// TIA Portal V17 export
// export: Created 2022-06-27T13:57:44.2303168Z, ExportSetting WithDefaults, DisplayName Totally Integrated Automation Portal, DisplayVersion V17 Update 3, DisplayName TIA Portal Openness, DisplayVersion V17 Update 3, DisplayName TIA Portal Version Control Interface, DisplayVersion V17, DisplayName SINAMICS Startdrive Advanced, DisplayVersion V17 Update1, DisplayName SINAMICS Startdrive G110M, G120, G120C, G120D, G120P, G115D, DisplayVersion V17 Update1, DisplayName SINAMICS Startdrive G130, G150, S120, S150, SINAMICS MV, S210, DisplayVersion V17 Update1, DisplayName STEP 7 Professional, DisplayVersion V17 Update 3, DisplayName STEP 7 Safety, DisplayVersion V17, DisplayName WinCC UA Professional, DisplayVersion V17 Update 3
FUNCTION_BLOCK "S041_DIRECT_START_MOTOR"   // FB41, LAD
{ S7_Optimized_Access := 'TRUE' }
VERSION : 0.1
// Info:
// -Motors that are named "Uxx-xx" instead of "Mxx-xx" use soft-starters
// stored: AutoNumber false, IsIECCheckEnabled false, IsRetainMemResEnabled false, MemoryReserve 100, SetENOAutomatically false, UDAEnableTagReadback false
   VAR
      ls_aDirect_Start_Motors : Bool;
      ls_aDriver_Motors : Bool;
      FB_INTERLOCKS_U33_2D { S7_SetPoint := 'True'} : "FB_INTERLOCKS";
      FB_MOTOR_DIRECT_START_U33_2D { S7_SetPoint := 'True'} : "FB_MOTOR_DIRECT_START";
      FB_INTERLOCKS_M33_4F { S7_SetPoint := 'True'} : "FB_INTERLOCKS";
      FB_MOTOR_DIRECT_START_M33_4F { S7_SetPoint := 'True'} : "FB_MOTOR_DIRECT_START";
      FB_INTERLOCKS_M33_6F { S7_SetPoint := 'True'} : "FB_INTERLOCKS";
      FB_MOTOR_DIRECT_START_M33_6F { S7_SetPoint := 'True'} : "FB_MOTOR_DIRECT_START";
      FB_INTERLOCKS_M35_2D { S7_SetPoint := 'True'} : "FB_INTERLOCKS";
      FB_MOTOR_DIRECT_START_M35_2D { S7_SetPoint := 'True'} : "FB_MOTOR_DIRECT_START";
      FB_MOTOR_DIRECT_START_U35_4D { S7_SetPoint := 'True'} : "FB_MOTOR_DIRECT_START";
      FB_INTERLOCKS_M36_5F { S7_SetPoint := 'True'} : "FB_INTERLOCKS";
      FB_MOTOR_DIRECT_START_M36_5F { S7_SetPoint := 'True'} : "FB_MOTOR_DIRECT_START";
      FB_INTERLOCKS_M36_7F { S7_SetPoint := 'True'} : "FB_INTERLOCKS";
      FB_MOTOR_DIRECT_START_M36_7F { S7_SetPoint := 'True'} : "FB_MOTOR_DIRECT_START";
      FB_INTERLOCKS_M36_9F { S7_SetPoint := 'True'} : "FB_INTERLOCKS";
      FB_MOTOR_DIRECT_START_M36_9F { S7_SetPoint := 'True'} : "FB_MOTOR_DIRECT_START";
      FB_INTERLOCKS_U37_2D { S7_SetPoint := 'True'} : "FB_INTERLOCKS";
      FB_MOTOR_DIRECT_START_U37_2D { S7_SetPoint := 'True'} : "FB_MOTOR_DIRECT_START";
      FB_INTERLOCKS_U37_3D { S7_SetPoint := 'True'} : "FB_INTERLOCKS";
      FB_MOTOR_DIRECT_START_U37_3D { S7_SetPoint := 'True'} : "FB_MOTOR_DIRECT_START";
      FB_INTERLOCKS_M37_5F { S7_SetPoint := 'True'} : "FB_INTERLOCKS";
      FB_MOTOR_DIRECT_START_M37_5F { S7_SetPoint := 'True'} : "FB_MOTOR_DIRECT_START";
      FB_INTERLOCKS_M37_7F { S7_SetPoint := 'True'} : "FB_INTERLOCKS";
      FB_MOTOR_DIRECT_START_M37_7F { S7_SetPoint := 'True'} : "FB_MOTOR_DIRECT_START";
      FB_INTERLOCKS_M37_9F { S7_SetPoint := 'True'} : "FB_INTERLOCKS";
      FB_MOTOR_DIRECT_START_M37_9F { S7_SetPoint := 'True'} : "FB_MOTOR_DIRECT_START";
      FB_INTERLOCKS_U35_4D { S7_SetPoint := 'True'} : "FB_INTERLOCKS";
   END_VAR
BEGIN

REGION Network 1: U33-2D - Burner Fan - Automatic on and off
END_REGION

REGION Network 2: U33-2D - Burner Fan - Interlocks
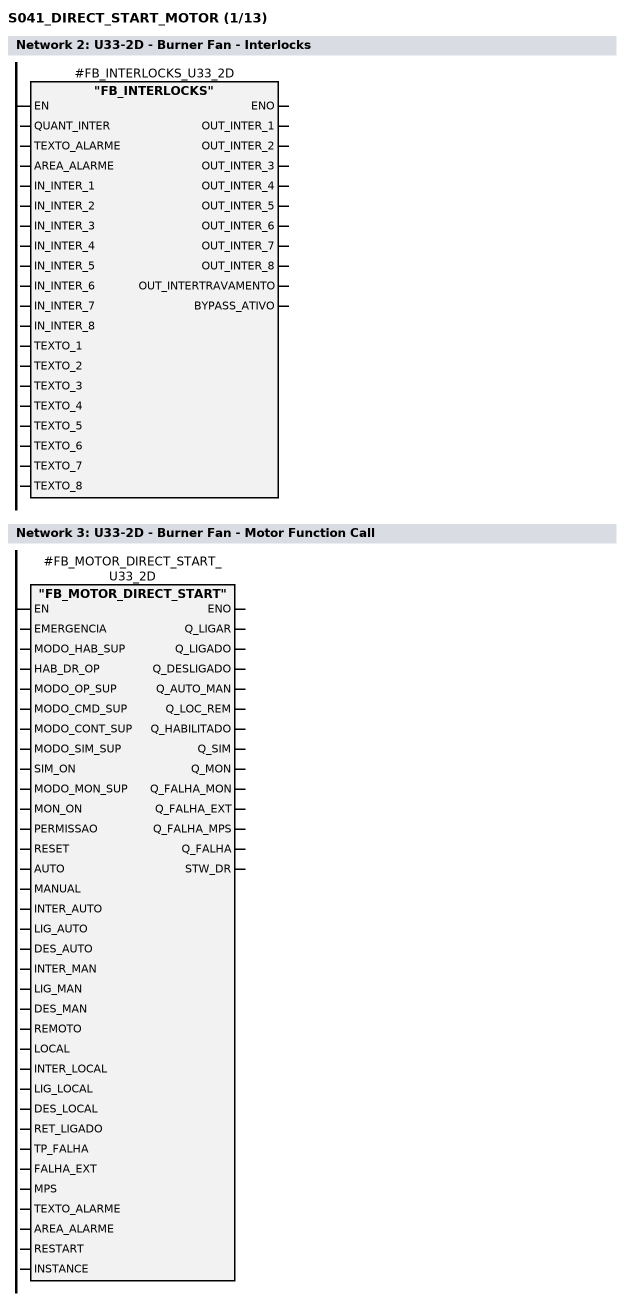
   RUNG wire#powerrail
      #FB_INTERLOCKS_U33_2D(QUANT_INTER :=, TEXTO_ALARME :=, AREA_ALARME :=, IN_INTER_1 :=, IN_INTER_2 :=, IN_INTER_3 :=, IN_INTER_4 :=, IN_INTER_5 :=, IN_INTER_6 :=, IN_INTER_7 :=, IN_INTER_8 :=, TEXTO_1 :=, TEXTO_2 :=, TEXTO_3 :=, TEXTO_4 :=, TEXTO_5 :=, TEXTO_6 :=, TEXTO_7 :=, TEXTO_8 :=, OUT_INTER_1 =>, OUT_INTER_2 =>, OUT_INTER_3 =>, OUT_INTER_4 =>, OUT_INTER_5 =>, OUT_INTER_6 =>, OUT_INTER_7 =>, OUT_INTER_8 =>, OUT_INTERTRAVAMENTO =>, BYPASS_ATIVO =>)
   END_RUNG
   // the same network as SCL:
   #FB_INTERLOCKS_U33_2D();   // "FB_INTERLOCKS"
END_REGION

REGION Network 3: U33-2D - Burner Fan - Motor Function Call
   RUNG wire#powerrail
      #FB_MOTOR_DIRECT_START_U33_2D(EMERGENCIA :=, MODO_HAB_SUP :=, HAB_DR_OP :=, MODO_OP_SUP :=, MODO_CMD_SUP :=, MODO_CONT_SUP :=, MODO_SIM_SUP :=, SIM_ON :=, MODO_MON_SUP :=, MON_ON :=, PERMISSAO :=, RESET :=, AUTO :=, MANUAL :=, INTER_AUTO :=, LIG_AUTO :=, DES_AUTO :=, INTER_MAN :=, LIG_MAN :=, DES_MAN :=, REMOTO :=, LOCAL :=, INTER_LOCAL :=, LIG_LOCAL :=, DES_LOCAL :=, RET_LIGADO :=, TP_FALHA :=, FALHA_EXT :=, MPS :=, TEXTO_ALARME :=, AREA_ALARME :=, RESTART :=, INSTANCE :=, Q_LIGAR =>, Q_LIGADO =>, Q_DESLIGADO =>, Q_AUTO_MAN =>, Q_LOC_REM =>, Q_HABILITADO =>, Q_SIM =>, Q_MON =>, Q_FALHA_MON =>, Q_FALHA_EXT =>, Q_FALHA_MPS =>, Q_FALHA =>, STW_DR =>)
   END_RUNG
   // the same network as SCL:
   #FB_MOTOR_DIRECT_START_U33_2D();   // "FB_MOTOR_DIRECT_START"
END_REGION

REGION Network 4: U33-2D - Burner Fan - Circuit Breaker
END_REGION

REGION Network 6: M33-4F - Rotary Valve Roaster Cyclone - Automatic on and off
END_REGION

REGION Network 7: M33-4F - Rotary Valve Roaster Cyclone - Interlocks
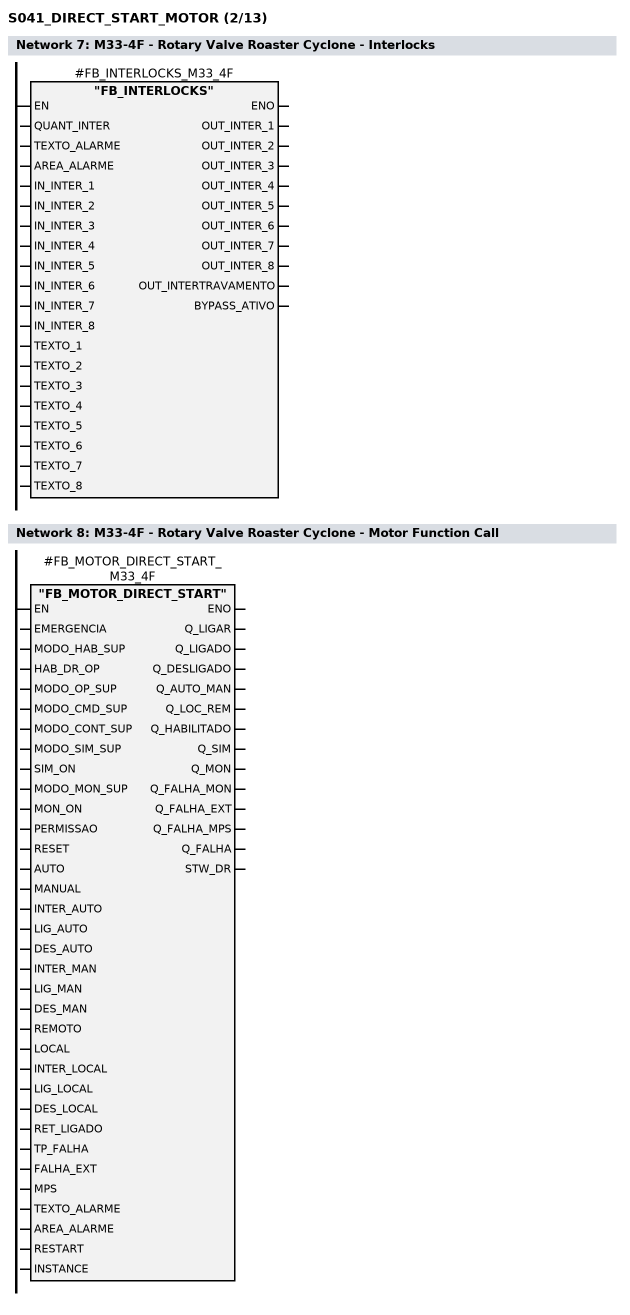
   RUNG wire#powerrail
      #FB_INTERLOCKS_M33_4F(QUANT_INTER :=, TEXTO_ALARME :=, AREA_ALARME :=, IN_INTER_1 :=, IN_INTER_2 :=, IN_INTER_3 :=, IN_INTER_4 :=, IN_INTER_5 :=, IN_INTER_6 :=, IN_INTER_7 :=, IN_INTER_8 :=, TEXTO_1 :=, TEXTO_2 :=, TEXTO_3 :=, TEXTO_4 :=, TEXTO_5 :=, TEXTO_6 :=, TEXTO_7 :=, TEXTO_8 :=, OUT_INTER_1 =>, OUT_INTER_2 =>, OUT_INTER_3 =>, OUT_INTER_4 =>, OUT_INTER_5 =>, OUT_INTER_6 =>, OUT_INTER_7 =>, OUT_INTER_8 =>, OUT_INTERTRAVAMENTO =>, BYPASS_ATIVO =>)
   END_RUNG
   // the same network as SCL:
   #FB_INTERLOCKS_M33_4F();   // "FB_INTERLOCKS"
END_REGION

REGION Network 8: M33-4F - Rotary Valve Roaster Cyclone - Motor Function Call
   RUNG wire#powerrail
      #FB_MOTOR_DIRECT_START_M33_4F(EMERGENCIA :=, MODO_HAB_SUP :=, HAB_DR_OP :=, MODO_OP_SUP :=, MODO_CMD_SUP :=, MODO_CONT_SUP :=, MODO_SIM_SUP :=, SIM_ON :=, MODO_MON_SUP :=, MON_ON :=, PERMISSAO :=, RESET :=, AUTO :=, MANUAL :=, INTER_AUTO :=, LIG_AUTO :=, DES_AUTO :=, INTER_MAN :=, LIG_MAN :=, DES_MAN :=, REMOTO :=, LOCAL :=, INTER_LOCAL :=, LIG_LOCAL :=, DES_LOCAL :=, RET_LIGADO :=, TP_FALHA :=, FALHA_EXT :=, MPS :=, TEXTO_ALARME :=, AREA_ALARME :=, RESTART :=, INSTANCE :=, Q_LIGAR =>, Q_LIGADO =>, Q_DESLIGADO =>, Q_AUTO_MAN =>, Q_LOC_REM =>, Q_HABILITADO =>, Q_SIM =>, Q_MON =>, Q_FALHA_MON =>, Q_FALHA_EXT =>, Q_FALHA_MPS =>, Q_FALHA =>, STW_DR =>)
   END_RUNG
   // the same network as SCL:
   #FB_MOTOR_DIRECT_START_M33_4F();   // "FB_MOTOR_DIRECT_START"
END_REGION

REGION Network 9: M33-4F - Rotary Valve Roaster Cyclone - Circuit Breaker
END_REGION

REGION Network 11: M33-6F - Water Pump - Automatic on and off
END_REGION

REGION Network 12: M33-6F - Water Pump - Interlocks
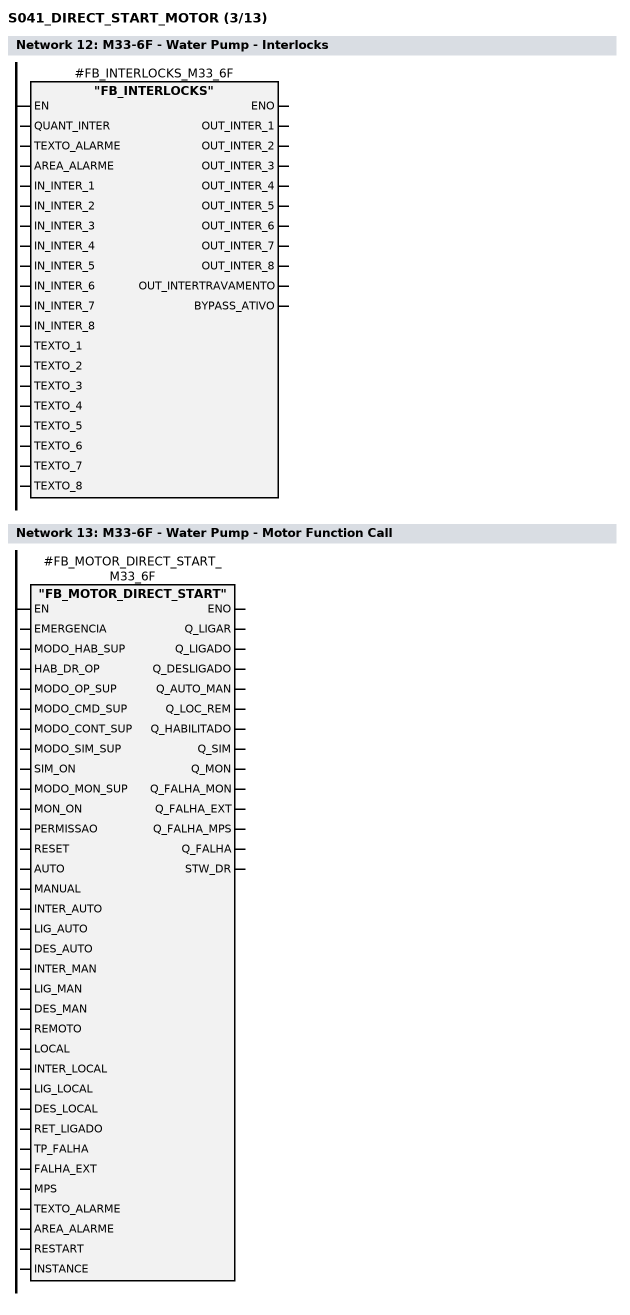
   RUNG wire#powerrail
      #FB_INTERLOCKS_M33_6F(QUANT_INTER :=, TEXTO_ALARME :=, AREA_ALARME :=, IN_INTER_1 :=, IN_INTER_2 :=, IN_INTER_3 :=, IN_INTER_4 :=, IN_INTER_5 :=, IN_INTER_6 :=, IN_INTER_7 :=, IN_INTER_8 :=, TEXTO_1 :=, TEXTO_2 :=, TEXTO_3 :=, TEXTO_4 :=, TEXTO_5 :=, TEXTO_6 :=, TEXTO_7 :=, TEXTO_8 :=, OUT_INTER_1 =>, OUT_INTER_2 =>, OUT_INTER_3 =>, OUT_INTER_4 =>, OUT_INTER_5 =>, OUT_INTER_6 =>, OUT_INTER_7 =>, OUT_INTER_8 =>, OUT_INTERTRAVAMENTO =>, BYPASS_ATIVO =>)
   END_RUNG
   // the same network as SCL:
   #FB_INTERLOCKS_M33_6F();   // "FB_INTERLOCKS"
END_REGION

REGION Network 13: M33-6F - Water Pump - Motor Function Call
   RUNG wire#powerrail
      #FB_MOTOR_DIRECT_START_M33_6F(EMERGENCIA :=, MODO_HAB_SUP :=, HAB_DR_OP :=, MODO_OP_SUP :=, MODO_CMD_SUP :=, MODO_CONT_SUP :=, MODO_SIM_SUP :=, SIM_ON :=, MODO_MON_SUP :=, MON_ON :=, PERMISSAO :=, RESET :=, AUTO :=, MANUAL :=, INTER_AUTO :=, LIG_AUTO :=, DES_AUTO :=, INTER_MAN :=, LIG_MAN :=, DES_MAN :=, REMOTO :=, LOCAL :=, INTER_LOCAL :=, LIG_LOCAL :=, DES_LOCAL :=, RET_LIGADO :=, TP_FALHA :=, FALHA_EXT :=, MPS :=, TEXTO_ALARME :=, AREA_ALARME :=, RESTART :=, INSTANCE :=, Q_LIGAR =>, Q_LIGADO =>, Q_DESLIGADO =>, Q_AUTO_MAN =>, Q_LOC_REM =>, Q_HABILITADO =>, Q_SIM =>, Q_MON =>, Q_FALHA_MON =>, Q_FALHA_EXT =>, Q_FALHA_MPS =>, Q_FALHA =>, STW_DR =>)
   END_RUNG
   // the same network as SCL:
   #FB_MOTOR_DIRECT_START_M33_6F();   // "FB_MOTOR_DIRECT_START"
END_REGION

REGION Network 14: M33-6F - Water Pump - Circuit Breaker
END_REGION

REGION Network 16: U35-2D - Roasting Chamber 1 - Automatic on and off
END_REGION

REGION Network 17: U35-2D - Roasting Chamber 1 - Interlocks
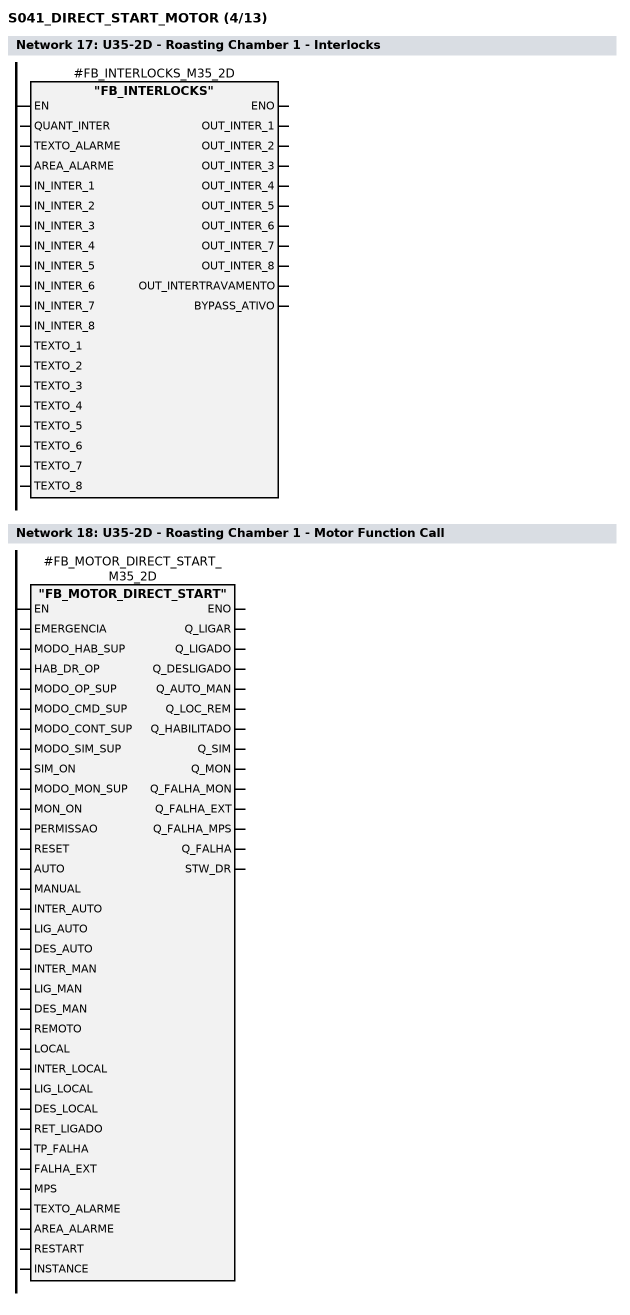
   RUNG wire#powerrail
      #FB_INTERLOCKS_M35_2D(QUANT_INTER :=, TEXTO_ALARME :=, AREA_ALARME :=, IN_INTER_1 :=, IN_INTER_2 :=, IN_INTER_3 :=, IN_INTER_4 :=, IN_INTER_5 :=, IN_INTER_6 :=, IN_INTER_7 :=, IN_INTER_8 :=, TEXTO_1 :=, TEXTO_2 :=, TEXTO_3 :=, TEXTO_4 :=, TEXTO_5 :=, TEXTO_6 :=, TEXTO_7 :=, TEXTO_8 :=, OUT_INTER_1 =>, OUT_INTER_2 =>, OUT_INTER_3 =>, OUT_INTER_4 =>, OUT_INTER_5 =>, OUT_INTER_6 =>, OUT_INTER_7 =>, OUT_INTER_8 =>, OUT_INTERTRAVAMENTO =>, BYPASS_ATIVO =>)
   END_RUNG
   // the same network as SCL:
   #FB_INTERLOCKS_M35_2D();   // "FB_INTERLOCKS"
END_REGION

REGION Network 18: U35-2D - Roasting Chamber 1 - Motor Function Call
   RUNG wire#powerrail
      #FB_MOTOR_DIRECT_START_M35_2D(EMERGENCIA :=, MODO_HAB_SUP :=, HAB_DR_OP :=, MODO_OP_SUP :=, MODO_CMD_SUP :=, MODO_CONT_SUP :=, MODO_SIM_SUP :=, SIM_ON :=, MODO_MON_SUP :=, MON_ON :=, PERMISSAO :=, RESET :=, AUTO :=, MANUAL :=, INTER_AUTO :=, LIG_AUTO :=, DES_AUTO :=, INTER_MAN :=, LIG_MAN :=, DES_MAN :=, REMOTO :=, LOCAL :=, INTER_LOCAL :=, LIG_LOCAL :=, DES_LOCAL :=, RET_LIGADO :=, TP_FALHA :=, FALHA_EXT :=, MPS :=, TEXTO_ALARME :=, AREA_ALARME :=, RESTART :=, INSTANCE :=, Q_LIGAR =>, Q_LIGADO =>, Q_DESLIGADO =>, Q_AUTO_MAN =>, Q_LOC_REM =>, Q_HABILITADO =>, Q_SIM =>, Q_MON =>, Q_FALHA_MON =>, Q_FALHA_EXT =>, Q_FALHA_MPS =>, Q_FALHA =>, STW_DR =>)
   END_RUNG
   // the same network as SCL:
   #FB_MOTOR_DIRECT_START_M35_2D();   // "FB_MOTOR_DIRECT_START"
END_REGION

REGION Network 19: U35-2D - Roasting Chamber 1 - Circuit Breaker
END_REGION

REGION Network 21: U35-4D - Roasting Chamber 2 - Automatic on and off
END_REGION

REGION Network 22: U35-4D - Roasting Chamber 2 - Interlocks
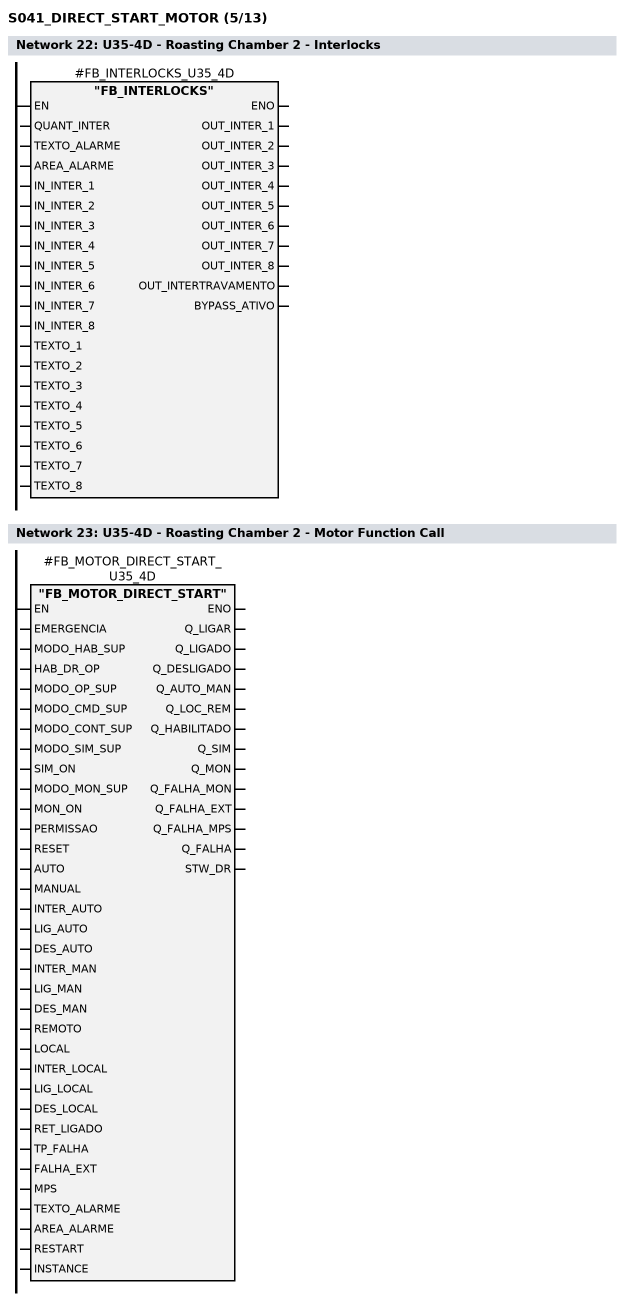
   RUNG wire#powerrail
      #FB_INTERLOCKS_U35_4D(QUANT_INTER :=, TEXTO_ALARME :=, AREA_ALARME :=, IN_INTER_1 :=, IN_INTER_2 :=, IN_INTER_3 :=, IN_INTER_4 :=, IN_INTER_5 :=, IN_INTER_6 :=, IN_INTER_7 :=, IN_INTER_8 :=, TEXTO_1 :=, TEXTO_2 :=, TEXTO_3 :=, TEXTO_4 :=, TEXTO_5 :=, TEXTO_6 :=, TEXTO_7 :=, TEXTO_8 :=, OUT_INTER_1 =>, OUT_INTER_2 =>, OUT_INTER_3 =>, OUT_INTER_4 =>, OUT_INTER_5 =>, OUT_INTER_6 =>, OUT_INTER_7 =>, OUT_INTER_8 =>, OUT_INTERTRAVAMENTO =>, BYPASS_ATIVO =>)
   END_RUNG
   // the same network as SCL:
   #FB_INTERLOCKS_U35_4D();   // "FB_INTERLOCKS"
END_REGION

REGION Network 23: U35-4D - Roasting Chamber 2 - Motor Function Call
   RUNG wire#powerrail
      #FB_MOTOR_DIRECT_START_U35_4D(EMERGENCIA :=, MODO_HAB_SUP :=, HAB_DR_OP :=, MODO_OP_SUP :=, MODO_CMD_SUP :=, MODO_CONT_SUP :=, MODO_SIM_SUP :=, SIM_ON :=, MODO_MON_SUP :=, MON_ON :=, PERMISSAO :=, RESET :=, AUTO :=, MANUAL :=, INTER_AUTO :=, LIG_AUTO :=, DES_AUTO :=, INTER_MAN :=, LIG_MAN :=, DES_MAN :=, REMOTO :=, LOCAL :=, INTER_LOCAL :=, LIG_LOCAL :=, DES_LOCAL :=, RET_LIGADO :=, TP_FALHA :=, FALHA_EXT :=, MPS :=, TEXTO_ALARME :=, AREA_ALARME :=, RESTART :=, INSTANCE :=, Q_LIGAR =>, Q_LIGADO =>, Q_DESLIGADO =>, Q_AUTO_MAN =>, Q_LOC_REM =>, Q_HABILITADO =>, Q_SIM =>, Q_MON =>, Q_FALHA_MON =>, Q_FALHA_EXT =>, Q_FALHA_MPS =>, Q_FALHA =>, STW_DR =>)
   END_RUNG
   // the same network as SCL:
   #FB_MOTOR_DIRECT_START_U35_4D();   // "FB_MOTOR_DIRECT_START"
END_REGION

REGION Network 24: U35-4D - Roasting Chamber 2 - Circuit Breaker
END_REGION

REGION Network 26: M36-5F - Rotary Valve Cooler Cyclone - Automatic on and off
END_REGION

REGION Network 27: M36-5F - Rotary Valve Cooler Cyclone - Interlocks
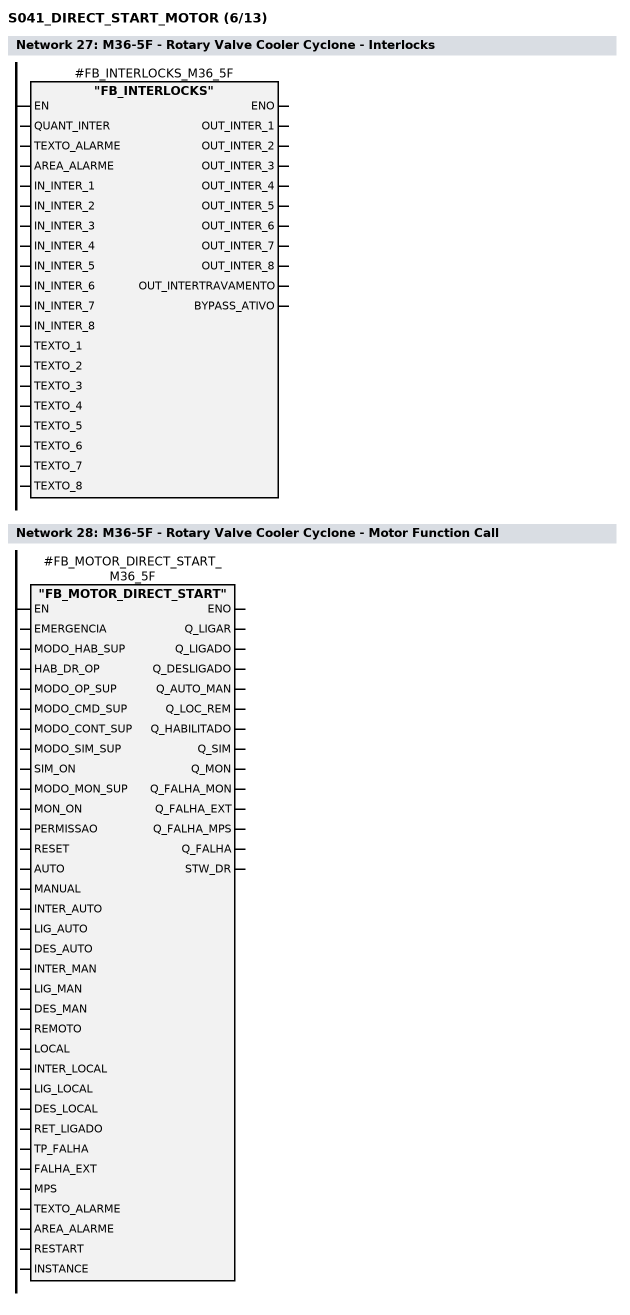
   RUNG wire#powerrail
      #FB_INTERLOCKS_M36_5F(QUANT_INTER :=, TEXTO_ALARME :=, AREA_ALARME :=, IN_INTER_1 :=, IN_INTER_2 :=, IN_INTER_3 :=, IN_INTER_4 :=, IN_INTER_5 :=, IN_INTER_6 :=, IN_INTER_7 :=, IN_INTER_8 :=, TEXTO_1 :=, TEXTO_2 :=, TEXTO_3 :=, TEXTO_4 :=, TEXTO_5 :=, TEXTO_6 :=, TEXTO_7 :=, TEXTO_8 :=, OUT_INTER_1 =>, OUT_INTER_2 =>, OUT_INTER_3 =>, OUT_INTER_4 =>, OUT_INTER_5 =>, OUT_INTER_6 =>, OUT_INTER_7 =>, OUT_INTER_8 =>, OUT_INTERTRAVAMENTO =>, BYPASS_ATIVO =>)
   END_RUNG
   // the same network as SCL:
   #FB_INTERLOCKS_M36_5F();   // "FB_INTERLOCKS"
END_REGION

REGION Network 28: M36-5F - Rotary Valve Cooler Cyclone - Motor Function Call
   RUNG wire#powerrail
      #FB_MOTOR_DIRECT_START_M36_5F(EMERGENCIA :=, MODO_HAB_SUP :=, HAB_DR_OP :=, MODO_OP_SUP :=, MODO_CMD_SUP :=, MODO_CONT_SUP :=, MODO_SIM_SUP :=, SIM_ON :=, MODO_MON_SUP :=, MON_ON :=, PERMISSAO :=, RESET :=, AUTO :=, MANUAL :=, INTER_AUTO :=, LIG_AUTO :=, DES_AUTO :=, INTER_MAN :=, LIG_MAN :=, DES_MAN :=, REMOTO :=, LOCAL :=, INTER_LOCAL :=, LIG_LOCAL :=, DES_LOCAL :=, RET_LIGADO :=, TP_FALHA :=, FALHA_EXT :=, MPS :=, TEXTO_ALARME :=, AREA_ALARME :=, RESTART :=, INSTANCE :=, Q_LIGAR =>, Q_LIGADO =>, Q_DESLIGADO =>, Q_AUTO_MAN =>, Q_LOC_REM =>, Q_HABILITADO =>, Q_SIM =>, Q_MON =>, Q_FALHA_MON =>, Q_FALHA_EXT =>, Q_FALHA_MPS =>, Q_FALHA =>, STW_DR =>)
   END_RUNG
   // the same network as SCL:
   #FB_MOTOR_DIRECT_START_M36_5F();   // "FB_MOTOR_DIRECT_START"
END_REGION

REGION Network 29: M36-5F - Rotary Valve Cooler Cyclone - Circuit Breaker
END_REGION

REGION Network 31: M36-7F - Cooler Conveyor Belt - Automatic on and off
END_REGION

REGION Network 32: M36-7F - Cooler Conveyor Belt - Interlocks
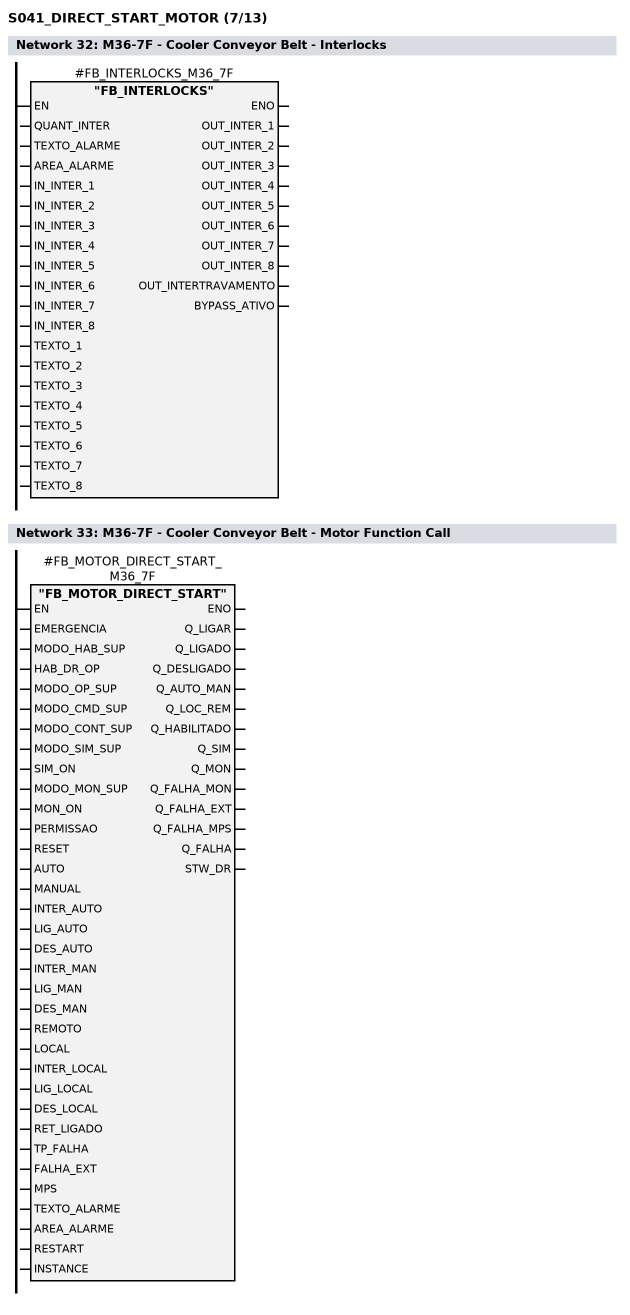
   RUNG wire#powerrail
      #FB_INTERLOCKS_M36_7F(QUANT_INTER :=, TEXTO_ALARME :=, AREA_ALARME :=, IN_INTER_1 :=, IN_INTER_2 :=, IN_INTER_3 :=, IN_INTER_4 :=, IN_INTER_5 :=, IN_INTER_6 :=, IN_INTER_7 :=, IN_INTER_8 :=, TEXTO_1 :=, TEXTO_2 :=, TEXTO_3 :=, TEXTO_4 :=, TEXTO_5 :=, TEXTO_6 :=, TEXTO_7 :=, TEXTO_8 :=, OUT_INTER_1 =>, OUT_INTER_2 =>, OUT_INTER_3 =>, OUT_INTER_4 =>, OUT_INTER_5 =>, OUT_INTER_6 =>, OUT_INTER_7 =>, OUT_INTER_8 =>, OUT_INTERTRAVAMENTO =>, BYPASS_ATIVO =>)
   END_RUNG
   // the same network as SCL:
   #FB_INTERLOCKS_M36_7F();   // "FB_INTERLOCKS"
END_REGION

REGION Network 33: M36-7F - Cooler Conveyor Belt - Motor Function Call
   RUNG wire#powerrail
      #FB_MOTOR_DIRECT_START_M36_7F(EMERGENCIA :=, MODO_HAB_SUP :=, HAB_DR_OP :=, MODO_OP_SUP :=, MODO_CMD_SUP :=, MODO_CONT_SUP :=, MODO_SIM_SUP :=, SIM_ON :=, MODO_MON_SUP :=, MON_ON :=, PERMISSAO :=, RESET :=, AUTO :=, MANUAL :=, INTER_AUTO :=, LIG_AUTO :=, DES_AUTO :=, INTER_MAN :=, LIG_MAN :=, DES_MAN :=, REMOTO :=, LOCAL :=, INTER_LOCAL :=, LIG_LOCAL :=, DES_LOCAL :=, RET_LIGADO :=, TP_FALHA :=, FALHA_EXT :=, MPS :=, TEXTO_ALARME :=, AREA_ALARME :=, RESTART :=, INSTANCE :=, Q_LIGAR =>, Q_LIGADO =>, Q_DESLIGADO =>, Q_AUTO_MAN =>, Q_LOC_REM =>, Q_HABILITADO =>, Q_SIM =>, Q_MON =>, Q_FALHA_MON =>, Q_FALHA_EXT =>, Q_FALHA_MPS =>, Q_FALHA =>, STW_DR =>)
   END_RUNG
   // the same network as SCL:
   #FB_MOTOR_DIRECT_START_M36_7F();   // "FB_MOTOR_DIRECT_START"
END_REGION

REGION Network 34: M36-7F - Cooler Conveyor Belt - Circuit Breaker
END_REGION

REGION Network 36: M36-9F - Tilted Conveyor Belt - Automatic on and off
END_REGION

REGION Network 37: M36-9F - Tilted Conveyor Belt - Interlocks
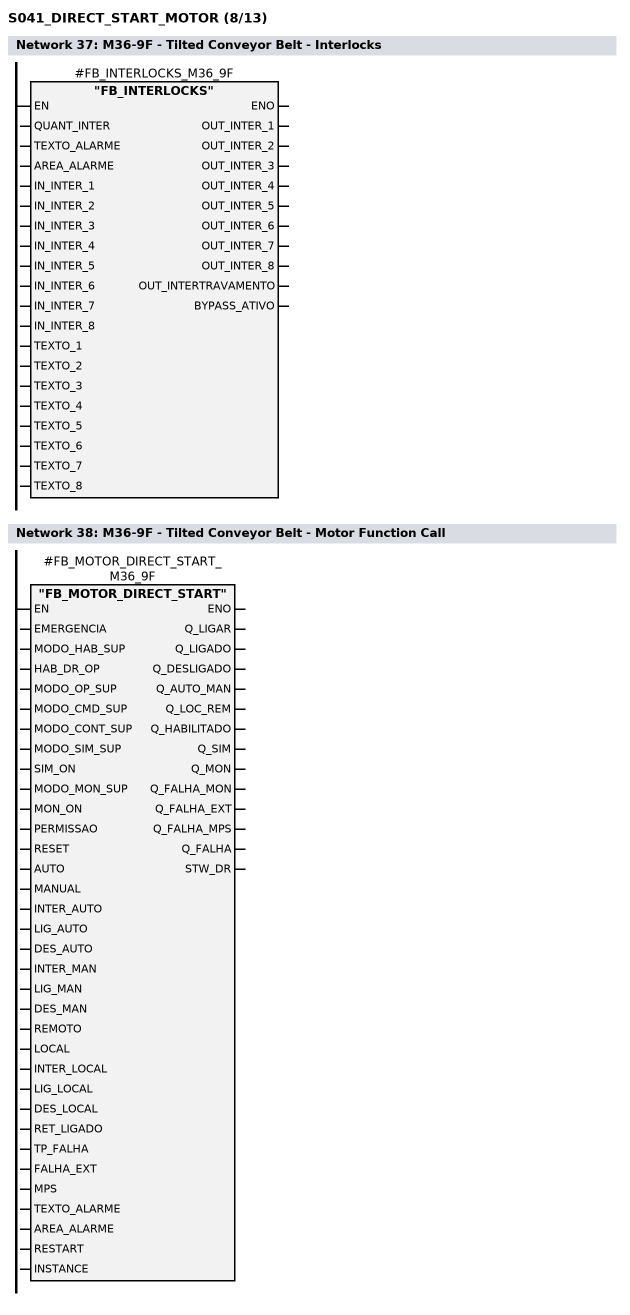
   RUNG wire#powerrail
      #FB_INTERLOCKS_M36_9F(QUANT_INTER :=, TEXTO_ALARME :=, AREA_ALARME :=, IN_INTER_1 :=, IN_INTER_2 :=, IN_INTER_3 :=, IN_INTER_4 :=, IN_INTER_5 :=, IN_INTER_6 :=, IN_INTER_7 :=, IN_INTER_8 :=, TEXTO_1 :=, TEXTO_2 :=, TEXTO_3 :=, TEXTO_4 :=, TEXTO_5 :=, TEXTO_6 :=, TEXTO_7 :=, TEXTO_8 :=, OUT_INTER_1 =>, OUT_INTER_2 =>, OUT_INTER_3 =>, OUT_INTER_4 =>, OUT_INTER_5 =>, OUT_INTER_6 =>, OUT_INTER_7 =>, OUT_INTER_8 =>, OUT_INTERTRAVAMENTO =>, BYPASS_ATIVO =>)
   END_RUNG
   // the same network as SCL:
   #FB_INTERLOCKS_M36_9F();   // "FB_INTERLOCKS"
END_REGION

REGION Network 38: M36-9F - Tilted Conveyor Belt - Motor Function Call
   RUNG wire#powerrail
      #FB_MOTOR_DIRECT_START_M36_9F(EMERGENCIA :=, MODO_HAB_SUP :=, HAB_DR_OP :=, MODO_OP_SUP :=, MODO_CMD_SUP :=, MODO_CONT_SUP :=, MODO_SIM_SUP :=, SIM_ON :=, MODO_MON_SUP :=, MON_ON :=, PERMISSAO :=, RESET :=, AUTO :=, MANUAL :=, INTER_AUTO :=, LIG_AUTO :=, DES_AUTO :=, INTER_MAN :=, LIG_MAN :=, DES_MAN :=, REMOTO :=, LOCAL :=, INTER_LOCAL :=, LIG_LOCAL :=, DES_LOCAL :=, RET_LIGADO :=, TP_FALHA :=, FALHA_EXT :=, MPS :=, TEXTO_ALARME :=, AREA_ALARME :=, RESTART :=, INSTANCE :=, Q_LIGAR =>, Q_LIGADO =>, Q_DESLIGADO =>, Q_AUTO_MAN =>, Q_LOC_REM =>, Q_HABILITADO =>, Q_SIM =>, Q_MON =>, Q_FALHA_MON =>, Q_FALHA_EXT =>, Q_FALHA_MPS =>, Q_FALHA =>, STW_DR =>)
   END_RUNG
   // the same network as SCL:
   #FB_MOTOR_DIRECT_START_M36_9F();   // "FB_MOTOR_DIRECT_START"
END_REGION

REGION Network 39: M36-9F - Tilted Conveyor Belt - Circuit Breaker
END_REGION

REGION Network 41: U37-2D - Cooler Chamber 1 - Automatic on and off
END_REGION

REGION Network 42: U37-2D - Cooler Chamber 1 - Interlocks
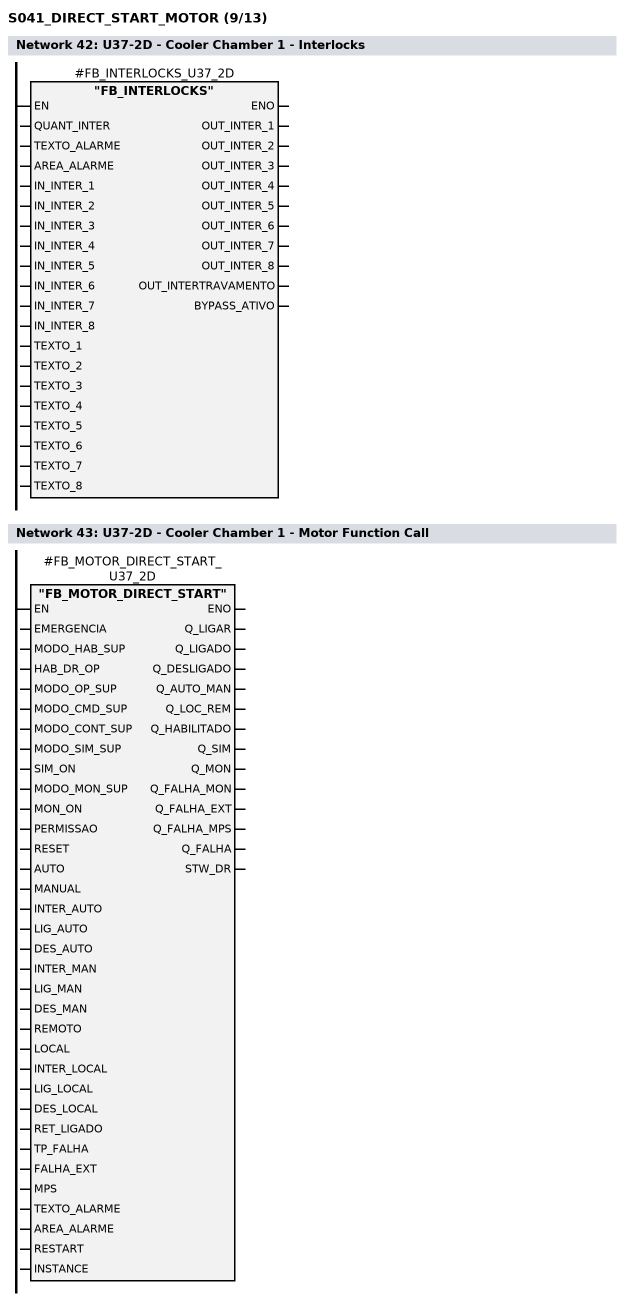
   RUNG wire#powerrail
      #FB_INTERLOCKS_U37_2D(QUANT_INTER :=, TEXTO_ALARME :=, AREA_ALARME :=, IN_INTER_1 :=, IN_INTER_2 :=, IN_INTER_3 :=, IN_INTER_4 :=, IN_INTER_5 :=, IN_INTER_6 :=, IN_INTER_7 :=, IN_INTER_8 :=, TEXTO_1 :=, TEXTO_2 :=, TEXTO_3 :=, TEXTO_4 :=, TEXTO_5 :=, TEXTO_6 :=, TEXTO_7 :=, TEXTO_8 :=, OUT_INTER_1 =>, OUT_INTER_2 =>, OUT_INTER_3 =>, OUT_INTER_4 =>, OUT_INTER_5 =>, OUT_INTER_6 =>, OUT_INTER_7 =>, OUT_INTER_8 =>, OUT_INTERTRAVAMENTO =>, BYPASS_ATIVO =>)
   END_RUNG
   // the same network as SCL:
   #FB_INTERLOCKS_U37_2D();   // "FB_INTERLOCKS"
END_REGION

REGION Network 43: U37-2D - Cooler Chamber 1 - Motor Function Call
   RUNG wire#powerrail
      #FB_MOTOR_DIRECT_START_U37_2D(EMERGENCIA :=, MODO_HAB_SUP :=, HAB_DR_OP :=, MODO_OP_SUP :=, MODO_CMD_SUP :=, MODO_CONT_SUP :=, MODO_SIM_SUP :=, SIM_ON :=, MODO_MON_SUP :=, MON_ON :=, PERMISSAO :=, RESET :=, AUTO :=, MANUAL :=, INTER_AUTO :=, LIG_AUTO :=, DES_AUTO :=, INTER_MAN :=, LIG_MAN :=, DES_MAN :=, REMOTO :=, LOCAL :=, INTER_LOCAL :=, LIG_LOCAL :=, DES_LOCAL :=, RET_LIGADO :=, TP_FALHA :=, FALHA_EXT :=, MPS :=, TEXTO_ALARME :=, AREA_ALARME :=, RESTART :=, INSTANCE :=, Q_LIGAR =>, Q_LIGADO =>, Q_DESLIGADO =>, Q_AUTO_MAN =>, Q_LOC_REM =>, Q_HABILITADO =>, Q_SIM =>, Q_MON =>, Q_FALHA_MON =>, Q_FALHA_EXT =>, Q_FALHA_MPS =>, Q_FALHA =>, STW_DR =>)
   END_RUNG
   // the same network as SCL:
   #FB_MOTOR_DIRECT_START_U37_2D();   // "FB_MOTOR_DIRECT_START"
END_REGION

REGION Network 44: U37-2D - Cooler Chamber 1 - Circuit Breaker
END_REGION

REGION Network 46: U37-3D - Cooler Chamber 2 - Automatic on and off
END_REGION

REGION Network 47: U37-3D - Cooler Chamber 2 - Interlocks
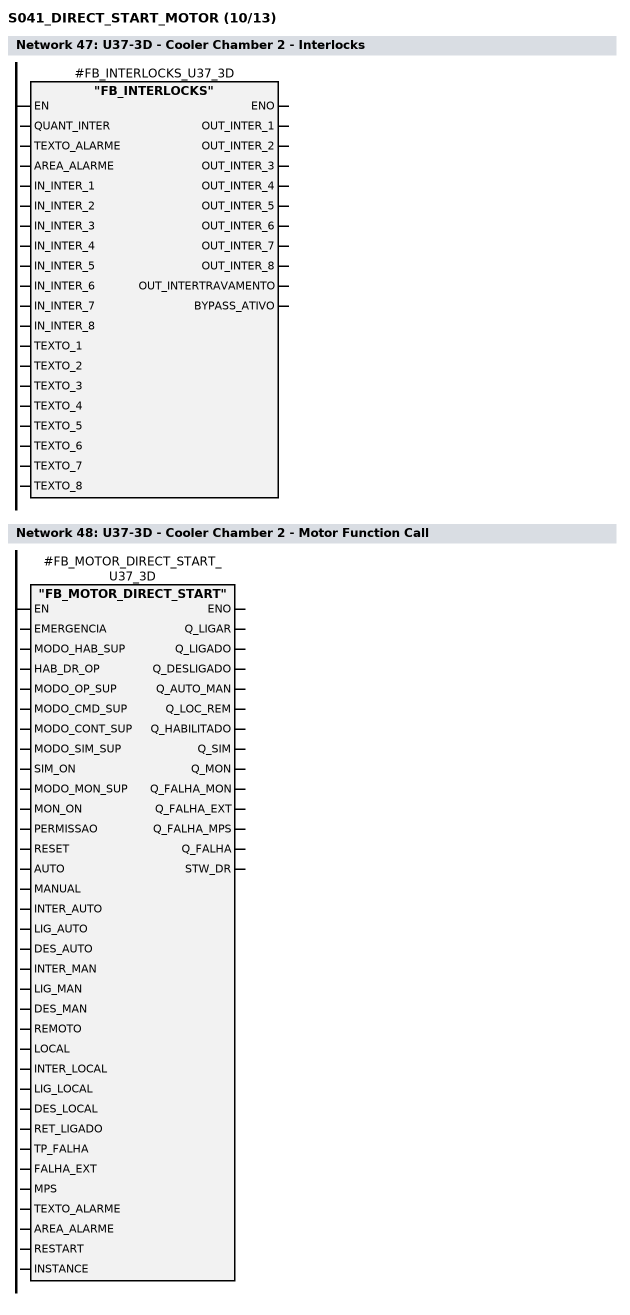
   RUNG wire#powerrail
      #FB_INTERLOCKS_U37_3D(QUANT_INTER :=, TEXTO_ALARME :=, AREA_ALARME :=, IN_INTER_1 :=, IN_INTER_2 :=, IN_INTER_3 :=, IN_INTER_4 :=, IN_INTER_5 :=, IN_INTER_6 :=, IN_INTER_7 :=, IN_INTER_8 :=, TEXTO_1 :=, TEXTO_2 :=, TEXTO_3 :=, TEXTO_4 :=, TEXTO_5 :=, TEXTO_6 :=, TEXTO_7 :=, TEXTO_8 :=, OUT_INTER_1 =>, OUT_INTER_2 =>, OUT_INTER_3 =>, OUT_INTER_4 =>, OUT_INTER_5 =>, OUT_INTER_6 =>, OUT_INTER_7 =>, OUT_INTER_8 =>, OUT_INTERTRAVAMENTO =>, BYPASS_ATIVO =>)
   END_RUNG
   // the same network as SCL:
   #FB_INTERLOCKS_U37_3D();   // "FB_INTERLOCKS"
END_REGION

REGION Network 48: U37-3D - Cooler Chamber 2 - Motor Function Call
   RUNG wire#powerrail
      #FB_MOTOR_DIRECT_START_U37_3D(EMERGENCIA :=, MODO_HAB_SUP :=, HAB_DR_OP :=, MODO_OP_SUP :=, MODO_CMD_SUP :=, MODO_CONT_SUP :=, MODO_SIM_SUP :=, SIM_ON :=, MODO_MON_SUP :=, MON_ON :=, PERMISSAO :=, RESET :=, AUTO :=, MANUAL :=, INTER_AUTO :=, LIG_AUTO :=, DES_AUTO :=, INTER_MAN :=, LIG_MAN :=, DES_MAN :=, REMOTO :=, LOCAL :=, INTER_LOCAL :=, LIG_LOCAL :=, DES_LOCAL :=, RET_LIGADO :=, TP_FALHA :=, FALHA_EXT :=, MPS :=, TEXTO_ALARME :=, AREA_ALARME :=, RESTART :=, INSTANCE :=, Q_LIGAR =>, Q_LIGADO =>, Q_DESLIGADO =>, Q_AUTO_MAN =>, Q_LOC_REM =>, Q_HABILITADO =>, Q_SIM =>, Q_MON =>, Q_FALHA_MON =>, Q_FALHA_EXT =>, Q_FALHA_MPS =>, Q_FALHA =>, STW_DR =>)
   END_RUNG
   // the same network as SCL:
   #FB_MOTOR_DIRECT_START_U37_3D();   // "FB_MOTOR_DIRECT_START"
END_REGION

REGION Network 49: U37-3D - Cooler Chamber 2 - Circuit Breaker
END_REGION

REGION Network 51: M37-5F - Rotary Valve Drying Chamber 1 Cyclone - Automatic on and off
END_REGION

REGION Network 52: M37-5F - Rotary Valve Drying Chamber 1 Cyclone - Interlocks
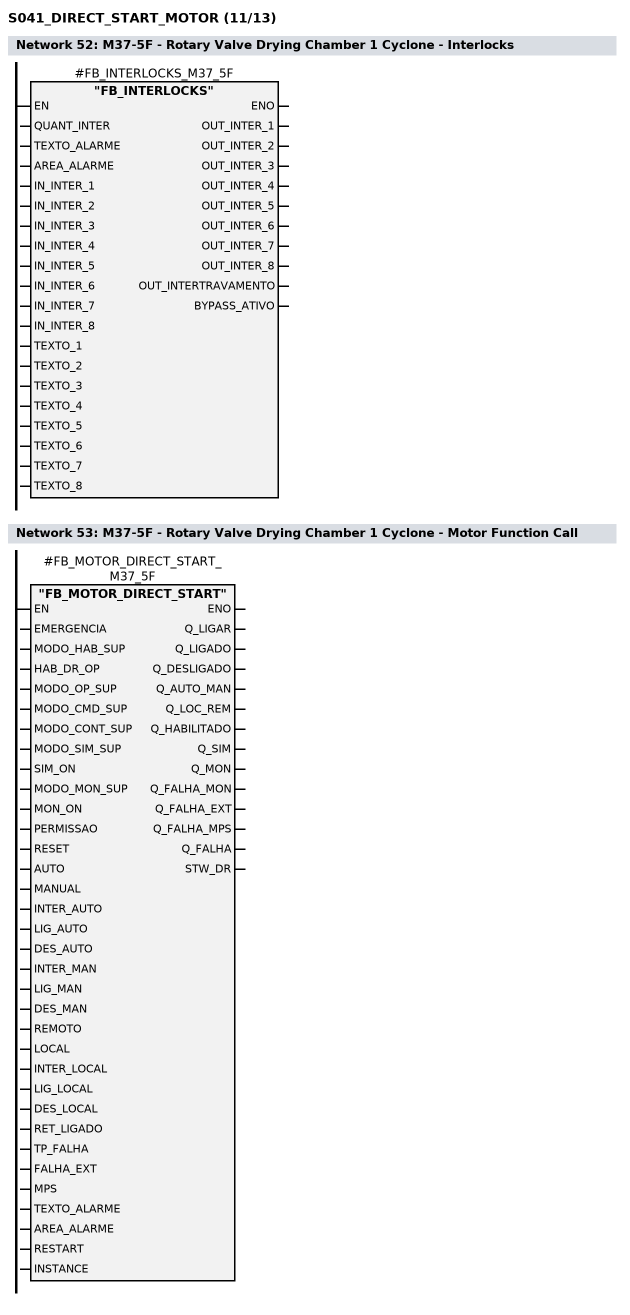
   RUNG wire#powerrail
      #FB_INTERLOCKS_M37_5F(QUANT_INTER :=, TEXTO_ALARME :=, AREA_ALARME :=, IN_INTER_1 :=, IN_INTER_2 :=, IN_INTER_3 :=, IN_INTER_4 :=, IN_INTER_5 :=, IN_INTER_6 :=, IN_INTER_7 :=, IN_INTER_8 :=, TEXTO_1 :=, TEXTO_2 :=, TEXTO_3 :=, TEXTO_4 :=, TEXTO_5 :=, TEXTO_6 :=, TEXTO_7 :=, TEXTO_8 :=, OUT_INTER_1 =>, OUT_INTER_2 =>, OUT_INTER_3 =>, OUT_INTER_4 =>, OUT_INTER_5 =>, OUT_INTER_6 =>, OUT_INTER_7 =>, OUT_INTER_8 =>, OUT_INTERTRAVAMENTO =>, BYPASS_ATIVO =>)
   END_RUNG
   // the same network as SCL:
   #FB_INTERLOCKS_M37_5F();   // "FB_INTERLOCKS"
END_REGION

REGION Network 53: M37-5F - Rotary Valve Drying Chamber 1 Cyclone - Motor Function Call
   RUNG wire#powerrail
      #FB_MOTOR_DIRECT_START_M37_5F(EMERGENCIA :=, MODO_HAB_SUP :=, HAB_DR_OP :=, MODO_OP_SUP :=, MODO_CMD_SUP :=, MODO_CONT_SUP :=, MODO_SIM_SUP :=, SIM_ON :=, MODO_MON_SUP :=, MON_ON :=, PERMISSAO :=, RESET :=, AUTO :=, MANUAL :=, INTER_AUTO :=, LIG_AUTO :=, DES_AUTO :=, INTER_MAN :=, LIG_MAN :=, DES_MAN :=, REMOTO :=, LOCAL :=, INTER_LOCAL :=, LIG_LOCAL :=, DES_LOCAL :=, RET_LIGADO :=, TP_FALHA :=, FALHA_EXT :=, MPS :=, TEXTO_ALARME :=, AREA_ALARME :=, RESTART :=, INSTANCE :=, Q_LIGAR =>, Q_LIGADO =>, Q_DESLIGADO =>, Q_AUTO_MAN =>, Q_LOC_REM =>, Q_HABILITADO =>, Q_SIM =>, Q_MON =>, Q_FALHA_MON =>, Q_FALHA_EXT =>, Q_FALHA_MPS =>, Q_FALHA =>, STW_DR =>)
   END_RUNG
   // the same network as SCL:
   #FB_MOTOR_DIRECT_START_M37_5F();   // "FB_MOTOR_DIRECT_START"
END_REGION

REGION Network 54: M37-5F - Rotary Valve Drying Chamber 1 Cyclone - Circuit Breaker
END_REGION

REGION Network 56: M37-7F - Rotary Valve Drying Chamber 2 Cyclone - Automatic on and off
END_REGION

REGION Network 57: M37-7F - Rotary Valve Drying Chamber 2 Cyclone - Interlocks
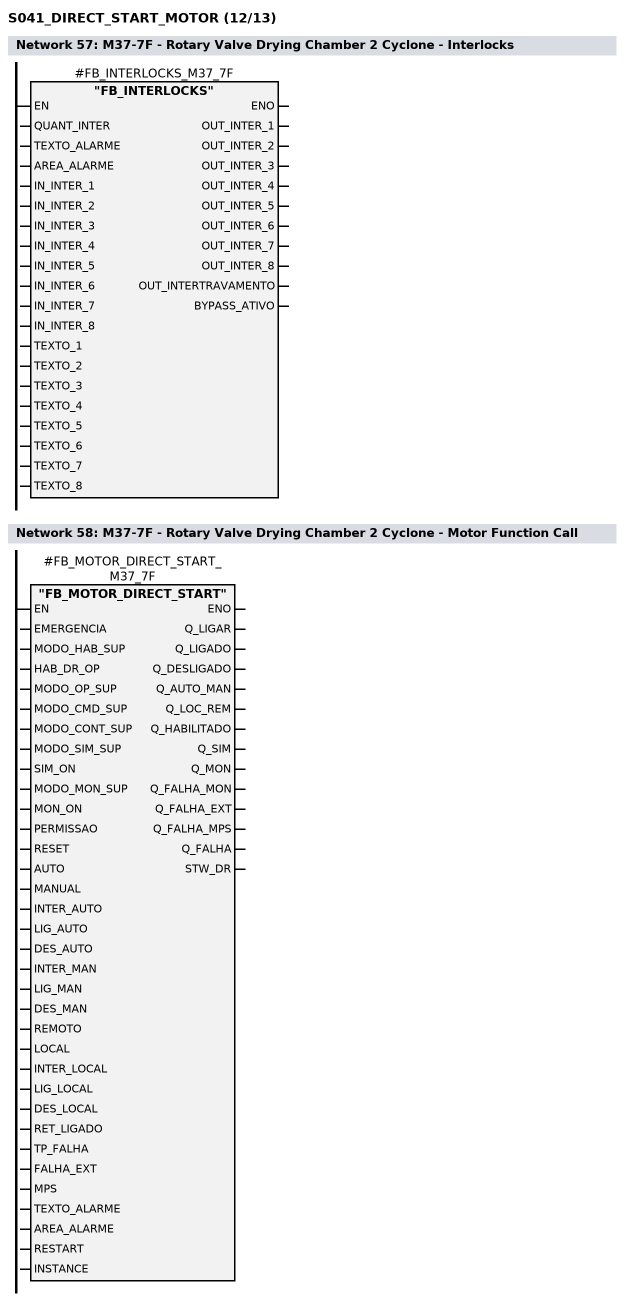
   RUNG wire#powerrail
      #FB_INTERLOCKS_M37_7F(QUANT_INTER :=, TEXTO_ALARME :=, AREA_ALARME :=, IN_INTER_1 :=, IN_INTER_2 :=, IN_INTER_3 :=, IN_INTER_4 :=, IN_INTER_5 :=, IN_INTER_6 :=, IN_INTER_7 :=, IN_INTER_8 :=, TEXTO_1 :=, TEXTO_2 :=, TEXTO_3 :=, TEXTO_4 :=, TEXTO_5 :=, TEXTO_6 :=, TEXTO_7 :=, TEXTO_8 :=, OUT_INTER_1 =>, OUT_INTER_2 =>, OUT_INTER_3 =>, OUT_INTER_4 =>, OUT_INTER_5 =>, OUT_INTER_6 =>, OUT_INTER_7 =>, OUT_INTER_8 =>, OUT_INTERTRAVAMENTO =>, BYPASS_ATIVO =>)
   END_RUNG
   // the same network as SCL:
   #FB_INTERLOCKS_M37_7F();   // "FB_INTERLOCKS"
END_REGION

REGION Network 58: M37-7F - Rotary Valve Drying Chamber 2 Cyclone - Motor Function Call
   RUNG wire#powerrail
      #FB_MOTOR_DIRECT_START_M37_7F(EMERGENCIA :=, MODO_HAB_SUP :=, HAB_DR_OP :=, MODO_OP_SUP :=, MODO_CMD_SUP :=, MODO_CONT_SUP :=, MODO_SIM_SUP :=, SIM_ON :=, MODO_MON_SUP :=, MON_ON :=, PERMISSAO :=, RESET :=, AUTO :=, MANUAL :=, INTER_AUTO :=, LIG_AUTO :=, DES_AUTO :=, INTER_MAN :=, LIG_MAN :=, DES_MAN :=, REMOTO :=, LOCAL :=, INTER_LOCAL :=, LIG_LOCAL :=, DES_LOCAL :=, RET_LIGADO :=, TP_FALHA :=, FALHA_EXT :=, MPS :=, TEXTO_ALARME :=, AREA_ALARME :=, RESTART :=, INSTANCE :=, Q_LIGAR =>, Q_LIGADO =>, Q_DESLIGADO =>, Q_AUTO_MAN =>, Q_LOC_REM =>, Q_HABILITADO =>, Q_SIM =>, Q_MON =>, Q_FALHA_MON =>, Q_FALHA_EXT =>, Q_FALHA_MPS =>, Q_FALHA =>, STW_DR =>)
   END_RUNG
   // the same network as SCL:
   #FB_MOTOR_DIRECT_START_M37_7F();   // "FB_MOTOR_DIRECT_START"
END_REGION

REGION Network 59: M37-7F - Rotary Valve Drying Chamber 2 Cyclone - Circuit Breaker
END_REGION

REGION Network 61: M37-9F - Cyclones Screw Conveyor - Automatic on and off
END_REGION

REGION Network 62: M37-9F - Cyclones Screw Conveyor - Interlocks
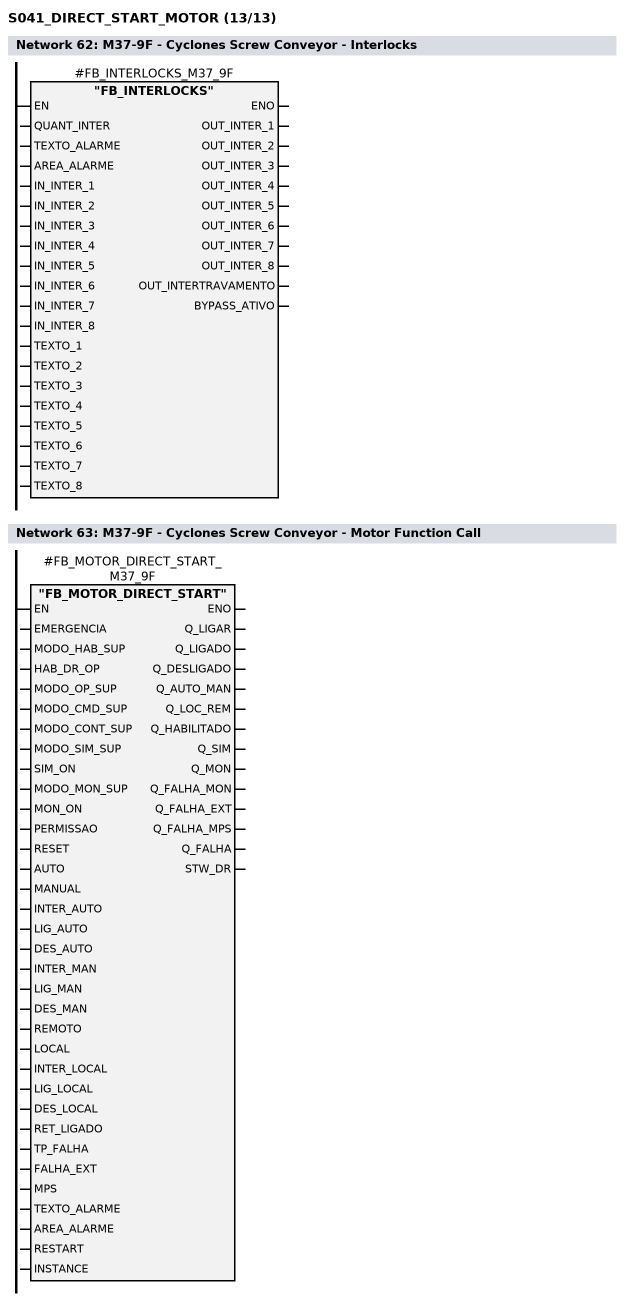
   RUNG wire#powerrail
      #FB_INTERLOCKS_M37_9F(QUANT_INTER :=, TEXTO_ALARME :=, AREA_ALARME :=, IN_INTER_1 :=, IN_INTER_2 :=, IN_INTER_3 :=, IN_INTER_4 :=, IN_INTER_5 :=, IN_INTER_6 :=, IN_INTER_7 :=, IN_INTER_8 :=, TEXTO_1 :=, TEXTO_2 :=, TEXTO_3 :=, TEXTO_4 :=, TEXTO_5 :=, TEXTO_6 :=, TEXTO_7 :=, TEXTO_8 :=, OUT_INTER_1 =>, OUT_INTER_2 =>, OUT_INTER_3 =>, OUT_INTER_4 =>, OUT_INTER_5 =>, OUT_INTER_6 =>, OUT_INTER_7 =>, OUT_INTER_8 =>, OUT_INTERTRAVAMENTO =>, BYPASS_ATIVO =>)
   END_RUNG
   // the same network as SCL:
   #FB_INTERLOCKS_M37_9F();   // "FB_INTERLOCKS"
END_REGION

REGION Network 63: M37-9F - Cyclones Screw Conveyor - Motor Function Call
   RUNG wire#powerrail
      #FB_MOTOR_DIRECT_START_M37_9F(EMERGENCIA :=, MODO_HAB_SUP :=, HAB_DR_OP :=, MODO_OP_SUP :=, MODO_CMD_SUP :=, MODO_CONT_SUP :=, MODO_SIM_SUP :=, SIM_ON :=, MODO_MON_SUP :=, MON_ON :=, PERMISSAO :=, RESET :=, AUTO :=, MANUAL :=, INTER_AUTO :=, LIG_AUTO :=, DES_AUTO :=, INTER_MAN :=, LIG_MAN :=, DES_MAN :=, REMOTO :=, LOCAL :=, INTER_LOCAL :=, LIG_LOCAL :=, DES_LOCAL :=, RET_LIGADO :=, TP_FALHA :=, FALHA_EXT :=, MPS :=, TEXTO_ALARME :=, AREA_ALARME :=, RESTART :=, INSTANCE :=, Q_LIGAR =>, Q_LIGADO =>, Q_DESLIGADO =>, Q_AUTO_MAN =>, Q_LOC_REM =>, Q_HABILITADO =>, Q_SIM =>, Q_MON =>, Q_FALHA_MON =>, Q_FALHA_EXT =>, Q_FALHA_MPS =>, Q_FALHA =>, STW_DR =>)
   END_RUNG
   // the same network as SCL:
   #FB_MOTOR_DIRECT_START_M37_9F();   // "FB_MOTOR_DIRECT_START"
END_REGION

REGION Network 64: M37-9F - Cyclones Screw Conveyor - Circuit Breaker
END_REGION
END_FUNCTION_BLOCK
